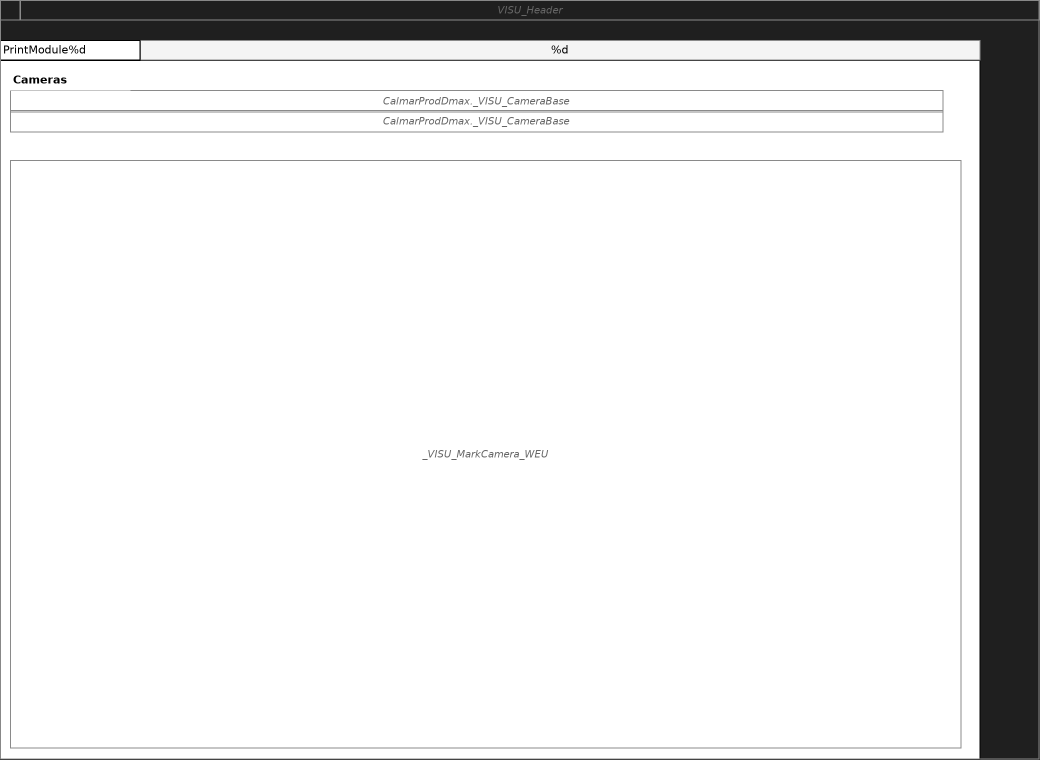
VISUALIZATION VISU_Cameras  // 1040x760
    Rectangle (0,60 980x700)
    Frame (10,160 951x588)
        shows _VISU_MarkCamera_WEU(mCam := PRG_PRINT.fbPrintModule[PRG_PRINT.fbModuleMaster.nViewPmSel].fbMarkCameraWeu, mMarkDetect := PRG_PRINT.fbPrintModule[PRG_PRINT.fbModuleMaster.nViewPmSel].fbMarkDetection)
    Frame (10,90 933x22)
        shows CalmarProdDmax._VISU_CameraBase(m_Inst := PRG_PRINT.fbPrintModule[PRG_PRINT.fbModuleMaster.nViewPmSel].fbNoCamera)
    Frame (10,110 933x22)
        shows CalmarProdDmax._VISU_CameraBase(m_Inst := PRG_PRINT.fbPrintModule[PRG_PRINT.fbModuleMaster.nViewPmSel].fbMarkCameraWeu)
    Scrollbar (140,40 840x20), "%d", text variable: PRG_PRINT.fbModuleMaster.nViewPmSel
        p1057716461: PRG_PRINT.fbModuleMaster.nViewPmSel
    Rectangle (0,40 140x20), "PrintModule%d", text variable: PRG_PRINT.fbModuleMaster.nViewPmSel
    Frame (20,0 1020x20)
        shows VISU_Header()
    Frame (0,0 20x20)
        shows VISU_ButtonBack()
    Rectangle (10,70 120x20), "Cameras"
END_VISUALIZATION

(* stored: Version 1.1.0.1, ProductVersion 3.1.4024.11
   Visu VISU_Cameras: Id {35356e6c-d44b-4d0e-b2f7-2e0dcd99e062} *)
